FUNCTION_BLOCK CENTRALConCTL (* Basic Function Block Type *)
  (* Standard: 61499-2 *)
  (* Version 0.2, 2003-12-04, JHC, Rockwell Automation, Renamed for better indexing. *)
  (* Version 0.1, 2002-11-05, JHC, Rockwell Automation, Corrected missing ST element in Algorithm REQ. *)
  (* Version 0.0, 2000-05-30, JHC, Rockwell Automation *)
  (* Compiler header: package fb.rt.cs725; *)
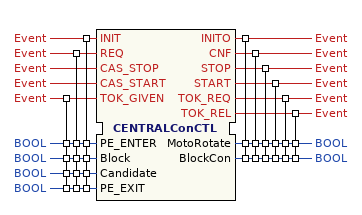
  EVENT_INPUT
    INIT WITH PE_ENTER, Block, Candidate, PE_EXIT; (* Initialization Request *)
    REQ WITH PE_ENTER, Block, Candidate, PE_EXIT; (* Normal Execution Request *)
    CAS_STOP;
    CAS_START;
    TOK_GIVEN WITH PE_ENTER, Block, PE_EXIT, Candidate;
  END_EVENT
  EVENT_OUTPUT
    INITO WITH MotoRotate, BlockCon; (* Initialization Confirm *)
    CNF WITH MotoRotate, BlockCon; (* Execution Confirmation *)
    STOP WITH MotoRotate, BlockCon;
    START WITH MotoRotate, BlockCon;
    TOK_REQ WITH MotoRotate, BlockCon;
    TOK_REL WITH MotoRotate, BlockCon;
  END_EVENT
  VAR_INPUT
    PE_ENTER : BOOL; (* Input event qualifier *)
    Block : BOOL;
    Candidate : BOOL;
    PE_EXIT : BOOL;
  END_VAR
  VAR_OUTPUT
    MotoRotate : BOOL; (* Output event qualifier *)
    BlockCon : BOOL;
  END_VAR
  VAR
    lastPE : BOOL := 1;
    lastBlock : BOOL := 0;
  END_VAR
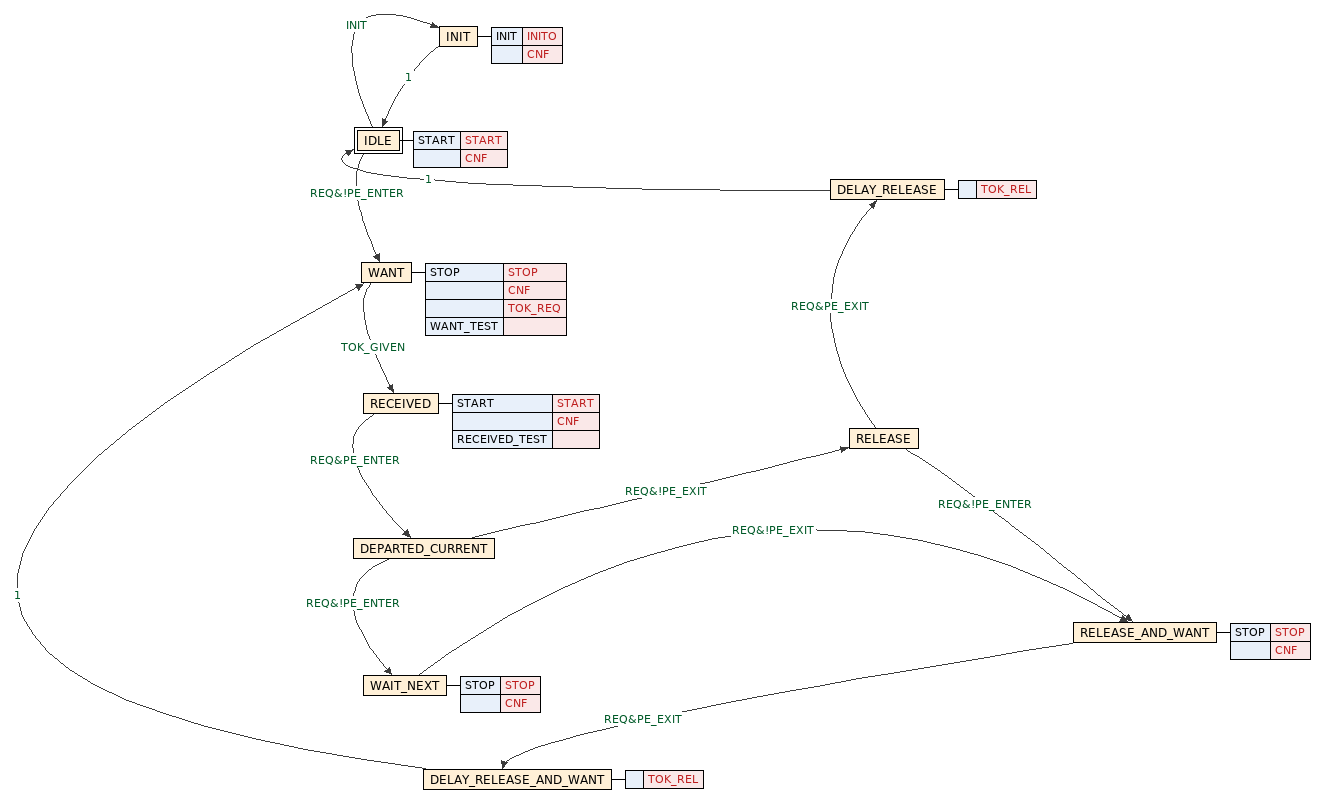
  EC_STATES
    IDLE : START -> START, -> CNF; (* Initial State *)
    INIT : INIT -> INITO, -> CNF; (* Initialization *)
    WANT : STOP -> STOP, -> CNF, -> TOK_REQ, WANT_TEST;
    RECEIVED : START -> START, -> CNF, RECEIVED_TEST;
    WAIT_NEXT : STOP -> STOP, -> CNF;
    DEPARTED_CURRENT;
    RELEASE;
    RELEASE_AND_WANT : STOP -> STOP, -> CNF;
    DELAY_RELEASE : -> TOK_REL;
    DELAY_RELEASE_AND_WANT : -> TOK_REL;
  END_STATES
  EC_TRANSITIONS
    IDLE TO INIT := INIT;
    INIT TO IDLE := 1;
    WANT TO RECEIVED := TOK_GIVEN;
    RECEIVED TO DEPARTED_CURRENT := REQ&PE_ENTER;
    DEPARTED_CURRENT TO WAIT_NEXT := REQ&!PE_ENTER;
    WAIT_NEXT TO RELEASE_AND_WANT := REQ&!PE_EXIT;
    DEPARTED_CURRENT TO RELEASE := REQ&!PE_EXIT;
    IDLE TO WANT := REQ&!PE_ENTER;
    DELAY_RELEASE TO IDLE := 1;
    RELEASE TO DELAY_RELEASE := REQ&PE_EXIT;
    DELAY_RELEASE_AND_WANT TO WANT := 1;
    RELEASE_AND_WANT TO DELAY_RELEASE_AND_WANT := REQ&PE_EXIT;
    RELEASE TO RELEASE_AND_WANT := REQ&!PE_ENTER;
  END_TRANSITIONS
  ALGORITHM INIT IN ST: (* Initialization algorithm *)
MotoRotate := TRUE;
Block := FALSE;

System.out.println(this + " " + MotoRotate);
System.out.println(MotoRotate);
  END_ALGORITHM
  ALGORITHM REQ IN ST: (* Normally executed algorithm *)
System.out.println(this +  " -> Candidate" + Candidate);
IF Candidate THEN
IF lastPE !:= PE_ENTER THEN
IF NOT PE_ENTER THEN
BlockCon:= TRUE;
System.out.println("BlockCon = true");
ELSE
BlockCon:=FALSE;
System.out.println("BlockCon = false");
END_IF
lastPE := PE_ENTER;
END_IF
IF lastBlock !:= Block THEN
IF Block THEN
STOP.serviceEvent(this);
MotoRotate := FALSE;
System.out.println("Cas Stop");
ELSE
START.serviceEvent(this);
MotoRotate := TRUE;
System.out.println("Cas Start");
END_IF
lastBlock := Block;
END_IF
END_IF
  END_ALGORITHM
  ALGORITHM START IN ST:
MotoRotate:=TRUE;
System.out.println(this + " Start " + MotoRotate);

System.out.println("Start " + MotoRotate);
  END_ALGORITHM
  ALGORITHM STOP IN ST:
MotoRotate := FALSE;
System.out.println(this + " Stop " + MotoRotate);

System.out.println("Stop " + MotoRotate);
  END_ALGORITHM
  ALGORITHM WANT_TEST IN Java:
System.out.println("IN WANTTTTTTTTTTTTTTTTTTTTTTTTTTT");
  END_ALGORITHM
  ALGORITHM RECEIVED_TEST IN Java:
System.out.println("RECEIVEDDDDD");
  END_ALGORITHM
END_FUNCTION_BLOCK
